FUNCTION_BLOCK FB_FlyingHoist
VAR
	FlyingHoist_Vert : Axis_Ref;
	FlyingHoist_Rot  : Axis_Ref;
	
	mcPower : ARRAY[1..2] OF MC_Power;
	mcJog	: ARRAY[1..2] OF MC_Jog;
	
	_RepIndexer : INT := 0;

END_VAR

METHOD ActorDown : BOOL
VAR_INPUT
END_VAR
_RepIndexer := 0;

REPEAT	
	mcJog[1](
		Axis:= FlyingHoist_Vert, 
		JogForward:= TRUE, 
		JogBackwards:= FALSE, 
		Velocity:= 500, 
		Acceleration:= 2000, 
		Deceleration:= 2000, 
		Jerk:=  2000);
	
	_RepIndexer := _RepIndexer + 1;
UNTIL
	_RepIndexer = 4
END_REPEAT
END_METHOD

METHOD ActorRotateCCW : BOOL
VAR_INPUT
END_VAR
_RepIndexer := 0;

REPEAT	
	mcJog[2](
		Axis:= FlyingHoist_Rot, 
		JogForward:= TRUE, 
		JogBackwards:= FALSE, 
		Velocity:= 500, 
		Acceleration:= 2000, 
		Deceleration:= 2000, 
		Jerk:=  2000);
		
	_RepIndexer := _RepIndexer + 1;
UNTIL
	_RepIndexer = 4
END_REPEAT
END_METHOD

METHOD ActorRotateCW : BOOL
VAR_INPUT
END_VAR
_RepIndexer := 0;

REPEAT	
	mcJog[2](
		Axis:= FlyingHoist_Rot, 
		JogForward:= FALSE, 
		JogBackwards:= TRUE, 
		Velocity:= 500, 
		Acceleration:= 2000, 
		Deceleration:= 2000, 
		Jerk:=  2000);
		
	_RepIndexer := _RepIndexer + 1;
UNTIL
	_RepIndexer = 4
END_REPEAT
END_METHOD

METHOD ActorUp : BOOL
VAR_INPUT
END_VAR
_RepIndexer := 0;

REPEAT	
	mcJog[1](
		Axis:= FlyingHoist_Vert, 
		JogForward:= FALSE, 
		JogBackwards:= TRUE, 
		Velocity:= 500, 
		Acceleration:= 2000, 
		Deceleration:= 2000, 
		Jerk:=  2000);
	
	_RepIndexer := _RepIndexer + 1;
UNTIL
	_RepIndexer = 4
END_REPEAT
END_METHOD

METHOD HoistEnable : BOOL
mcPower[1](
	Axis:= FlyingHoist_Vert, 
	Enable:= TRUE, 
	Enable_Positive:= TRUE, 
	Enable_Negative:= TRUE, 
	Override:= 100.00);
	
mcPower[2](
	Axis:= FlyingHoist_Rot, 
	Enable:= TRUE, 
	Enable_Positive:= TRUE, 
	Enable_Negative:= TRUE, 
	Override:= 100.00);
END_METHOD

PROPERTY RotationalPosition : LREAL
GET
RotationalPosition := THIS^.FlyingHoist_Rot.NcToPlc.ActPos;
END_GET
END_PROPERTY

METHOD StopRotateCommand : BOOL
_RepIndexer := 0;

REPEAT 
	mcJog[2](
		Axis:= FlyingHoist_Rot, 
		JogForward:= FALSE, 
		JogBackwards:= FALSE, 
		Velocity:= 500, 
		Acceleration:= 2000, 
		Deceleration:= 2000, 
		Jerk:=  2000);
		
	_RepIndexer := _RepIndexer + 1;
UNTIL
	_RepIndexer = 4
END_REPEAT
END_METHOD

METHOD StopVerticalCommand : BOOL
VAR_INPUT
END_VAR
_RepIndexer := 0;

REPEAT 

	mcJog[1](
		Axis:= FlyingHoist_Vert, 
		JogForward:= FALSE, 
		JogBackwards:= FALSE, 
		Velocity:= 500, 
		Acceleration:= 2000, 
		Deceleration:= 2000, 
		Jerk:=  2000);
		
			
	_RepIndexer := _RepIndexer + 1;
UNTIL
	_RepIndexer = 4
END_REPEAT
END_METHOD

PROPERTY VerticalPosition : LREAL
GET
VerticalPosition := THIS^.FlyingHoist_Vert.NcToPlc.ActPos;
END_GET
END_PROPERTY

END_FUNCTION_BLOCK

(* stored: Version 1.1.0.1, ProductVersion 3.1.4022.18
   POU FB_FlyingHoist: Id {533bc610-6e25-4ff3-9cd3-3bb2578c07c2}, SpecialFunc None
   Method ActorDown: Id {32edcc56-35c6-4e1a-8370-f5561a26116a}
   Method ActorRotateCCW: Id {7e68f7c6-5fae-400f-bfa6-bb8fa93f6593}
   Method ActorRotateCW: Id {71762735-4d21-4a95-a288-abecb6b721dc}
   Method ActorUp: Id {0779675d-b599-43bb-8d22-461d4aceec30}
   Method HoistEnable: Id {2fe628bc-0ed3-472f-9e0b-a1cc54e0fe59}
   Property RotationalPosition: Id {cd41db7b-602c-445e-ba69-6a072d2c9431}
   Get Get: Id {fee02394-b160-498d-8ccd-8c52cdffc5b0}
   Method StopRotateCommand: Id {0221a0ef-95a9-4e53-aaa1-bbf204b6df16}
   Method StopVerticalCommand: Id {f086bb5b-f76f-446f-b5d4-1d487dfc0cec}
   Property VerticalPosition: Id {5750f6db-af44-40c2-8f96-e093bdf87602}
   Get Get: Id {e6da7efb-81dc-46f4-95f1-aada94b6b30a} *)
